(* IEC 61131-3 sources: POMIRTS_lab3/AS/Library_2/AsNxDnS, 3 files *)

(* ---- AsNxDnS.typ ---- *)
TYPE

END_TYPE

(* ---- AsNxDnS.fun ---- *)
{REDUND_CONTEXT} {REDUND_UNREPLICABLE} FUNCTION_BLOCK nxdnsSubscribe			(*subscribe slave*)
	VAR_INPUT
		enable			: BOOL;			(*enables execution*)
		pDevice			: UDINT;		(*interface name given as a pointer, e.g., "SL<x>.SS<y>.IF<z>"*)
	END_VAR
	VAR
        _state			: UINT;			(*internal variable*)
		_result			: UINT;			(*internal variable*)
        _srcId			: UDINT;		(*internal variable*)
	END_VAR
	VAR_OUTPUT
		status			: UINT;			(*execution status: ERR_OK, ERR_FUB_ENABLE_FALSE, ERR_FUB_BUSY, 0xXXXX = see help*)
		dnStatus		: UDINT;		(*devicenet stack status*)
	END_VAR
END_FUNCTION_BLOCK

{REDUND_CONTEXT} {REDUND_UNREPLICABLE} FUNCTION_BLOCK nxdnsUnsubscribe			(*unsubscribe slave*)
	VAR_INPUT
		enable			: BOOL;			(*enables execution*)
		pDevice			: UDINT;		(*interface name given as a pointer, e.g., "SL<x>.SS<y>.IF<z>"*)
	END_VAR
	VAR
        _state			: UINT;			(*internal variable*)
		_result			: UINT;			(*internal variable*)
        _srcId			: UDINT;		(*internal variable*)
	END_VAR
	VAR_OUTPUT
		status			: UINT;			(*execution status: ERR_OK, ERR_FUB_ENABLE_FALSE, ERR_FUB_BUSY, 0xXXXX = see help*)
		dnStatus		: UDINT;		(*devicenet stack status*)
	END_VAR
END_FUNCTION_BLOCK

{REDUND_CONTEXT} {REDUND_UNREPLICABLE} FUNCTION_BLOCK nxdnsRegisterClass		(*register class ID*)
	VAR_INPUT
		enable			: BOOL;			(*enables execution*)
		pDevice			: UDINT;		(*interface name given as a pointer, e.g., "SL<x>.SS<y>.IF<z>"*)
		classId			: UDINT;		(*class designator*)
		accessType		: UDINT;		(*reserved unused, set to 0*)
	END_VAR
	VAR
        _state			: UINT;			(*internal variable*)
		_result			: UINT;			(*internal variable*)
        _srcId			: UDINT;		(*internal variable*)
	END_VAR
	VAR_OUTPUT
		status			: UINT;			(*execution status: ERR_OK, ERR_FUB_ENABLE_FALSE, ERR_FUB_BUSY, 0xXXXX = see help*)
		dnStatus		: UDINT;		(*devicenet stack status*)
	END_VAR
END_FUNCTION_BLOCK

{REDUND_CONTEXT} {REDUND_UNREPLICABLE} FUNCTION_BLOCK nxdnsUnregisterClass		(*unregister class ID*)
	VAR_INPUT
		enable			: BOOL;			(*enables execution*)
		pDevice			: UDINT;		(*interface name given as a pointer, e.g., "SL<x>.SS<y>.IF<z>"*)
		classId			: UDINT;		(*class designator*)
		accessType		: UDINT;		(*reserved unused, set to 0*)
	END_VAR
	VAR
        _state			: UINT;			(*internal variable*)
		_result			: UINT;			(*internal variable*)
        _srcId			: UDINT;		(*internal variable*)
	END_VAR
	VAR_OUTPUT
		status			: UINT;			(*execution status: ERR_OK, ERR_FUB_ENABLE_FALSE, ERR_FUB_BUSY, 0xXXXX = see help*)
		dnStatus		: UDINT;		(*devicenet stack status*)
	END_VAR
END_FUNCTION_BLOCK

{REDUND_CONTEXT} {REDUND_UNREPLICABLE} FUNCTION_BLOCK nxdnsGetAttributeInd		(*get attribute indication*)
	VAR_INPUT
		enable			: BOOL;			(*enables execution*)
		pDevice			: UDINT;		(*interface name given as a pointer, e.g., "SL<x>.SS<y>.IF<z>"*)
	END_VAR
	VAR
        _state			: UINT;			(*internal variable*)
		_result			: UINT;			(*internal variable*)
        _srcId			: UDINT;		(*internal variable*)
	END_VAR
	VAR_OUTPUT
		status			: UINT;			(*execution status: ERR_OK, ERR_FUB_ENABLE_FALSE, ERR_FUB_BUSY, 0xXXXX = see help*)
		dnStatus		: UDINT;		(*devicenet stack status*)
		source			: UDINT;		(*source*)
		sourceId		: UDINT;		(*source ID*)
		classId			: UINT;			(*class ID of user application object requested by master*)
		instanceId		: UINT;			(*instance ID of user application object requested by master*)
		attributeId		: UINT;			(*attribute ID of user application object requested by master*)
	END_VAR
END_FUNCTION_BLOCK

{REDUND_CONTEXT} {REDUND_UNREPLICABLE} FUNCTION_BLOCK nxdnsSetAttributeInd		(*set attribute indication*)
	VAR_INPUT
		enable			: BOOL;			(*enables execution*)
		pDevice			: UDINT;		(*interface name given as a pointer, e.g., "SL<x>.SS<y>.IF<z>"*)
		maxDataCount	: UDINT;		(*maximum data count*)
		pData			: UDINT;		(*information data buffer given as pointer*)
	END_VAR
	VAR
        _state			: UINT;			(*internal variable*)
		_result			: UINT;			(*internal variable*)
        _srcId			: UDINT;		(*internal variable*)
	END_VAR
	VAR_OUTPUT
		status			: UINT;			(*execution status: ERR_OK, ERR_FUB_ENABLE_FALSE, ERR_FUB_BUSY, 0xXXXX = see help*)
		dnStatus		: UDINT;		(*devicenet stack status*)
		source			: UDINT;		(*source*)
		sourceId		: UDINT;		(*source ID*)
		classId			: UINT;			(*class ID of user application object requested by master*)
		instanceId		: UINT;			(*instance ID of user application object requested by master*)
		attributeId		: UINT;			(*attribute ID of user application object requested by master*)
		dataCount		: UINT;			(*data count of bytes to be written by the user application*)
	END_VAR
END_FUNCTION_BLOCK

{REDUND_CONTEXT} {REDUND_UNREPLICABLE} FUNCTION_BLOCK nxdnsGetAttributeRes		(*get attribute response*)
	VAR_INPUT
		enable			: BOOL;			(*enables execution*)
		pDevice			: UDINT;		(*interface name given as a pointer, e.g., "SL<x>.SS<y>.IF<z>"*)
		source			: UDINT;		(*source*)
		sourceId		: UDINT;		(*source ID*)
		classId			: UINT;			(*class ID of user application object requested by master*)
		instanceId		: UINT;			(*instance ID of user application object requested by master*)
		attributeId		: UINT;			(*attribute ID of user application object requested by master*)
		dataCount		: UINT;			(*data count of bytes to be read by the user application*)
		generalError	: USINT;		(*general error code returned by the user, see help*)
		additionalError	: USINT;		(*additional error code, user specific*)
		pData			: UDINT;		(*information data buffer given as pointer*)
	END_VAR
	VAR
        _state			: UINT;			(*internal variable*)
		_result			: UINT;			(*internal variable*)
        _srcId			: UDINT;		(*internal variable*)
	END_VAR
	VAR_OUTPUT
		status			: UINT;			(*execution status: ERR_OK, ERR_FUB_ENABLE_FALSE, ERR_FUB_BUSY, 0xXXXX = see help*)
		dnStatus		: UDINT;		(*devicenet stack status*)
	END_VAR
END_FUNCTION_BLOCK

{REDUND_CONTEXT} {REDUND_UNREPLICABLE} FUNCTION_BLOCK nxdnsSetAttributeRes		(*set attribute response*)
	VAR_INPUT
		enable			: BOOL;			(*enables execution*)
		pDevice			: UDINT;		(*interface name given as a pointer, e.g., "SL<x>.SS<y>.IF<z>"*)
		source			: UDINT;		(*message source*)
		sourceId		: UDINT;		(*message source ID*)
		classId			: UINT;			(*class ID of user application object requested by master*)
		instanceId		: UINT;			(*instance ID of user application object requested by master*)
		attributeId		: UINT;			(*attribute ID of user application object requested by master*)
		dataCount		: UINT;			(*data count of bytes written by the user application*)
		generalError	: USINT;		(*general error code returned by the user, see help*)
		additionalError	: USINT;		(*additional error code, user specific*)
	END_VAR
	VAR
        _state			: UINT;			(*internal variable*)
		_result			: UINT;			(*internal variable*)
        _srcId			: UDINT;		(*internal variable*)
	END_VAR
	VAR_OUTPUT
		status			: UINT;			(*execution status: ERR_OK, ERR_FUB_ENABLE_FALSE, ERR_FUB_BUSY, 0xXXXX = see help*)
		dnStatus		: UDINT;		(*devicenet stack status*)
	END_VAR
END_FUNCTION_BLOCK

{REDUND_CONTEXT} {REDUND_UNREPLICABLE} FUNCTION_BLOCK nxdnsSetAdr				(*set address*)
	VAR_INPUT
		enable			: BOOL;			(*enables execution*)
		pDevice			: UDINT;		(*interface name given as a pointer, e.g., "SL<x>.SS<y>.IF<z>"*)
		address			: UDINT;		(*new slave address*)
	END_VAR
	VAR
        _state			: UINT;			(*internal variable*)
		_result			: UINT;			(*internal variable*)
        _srcId			: UDINT;		(*internal variable*)
	END_VAR
	VAR_OUTPUT
		status			: UINT;			(*execution status: ERR_OK, ERR_FUB_ENABLE_FALSE, ERR_FUB_BUSY, 0xXXXX = see help*)
		dnStatus		: UDINT;		(*devicenet stack status*)
	END_VAR
END_FUNCTION_BLOCK

{REDUND_CONTEXT} {REDUND_UNREPLICABLE} FUNCTION_BLOCK nxdnsStartBusComm		(*start bus communication*)
	VAR_INPUT
		enable			: BOOL;			(*enables execution*)
		pDevice			: UDINT;		(*interface name given as a pointer, e.g., "SL<x>.SS<y>.IF<z>"*)
	END_VAR
	VAR
        _state			: UINT;			(*internal variable*)
		_result			: UINT;			(*internal variable*)
        _srcId			: UDINT;		(*internal variable*)
	END_VAR
	VAR_OUTPUT
		status			: UINT;			(*execution status: ERR_OK, ERR_FUB_ENABLE_FALSE, ERR_FUB_BUSY, 0xXXXX = see help*)
		dnStatus		: UDINT;		(*devicenet stack status*)
	END_VAR
END_FUNCTION_BLOCK

(* ---- AsNxDnS.var ---- *)
VAR CONSTANT
	nxdnsERR_INVALID_DEVICE					: UINT	:= 35360;		(*error invalid device*)
	nxdnsERR_SEND_MESSAGE					: UINT	:= 35361;		(*error send message*)
	nxdnsERR_TIMEOUT						: UINT	:= 35362;		(*error timeout*)
	nxdnsERR_DEVICENET_STACK				: UINT	:= 35363;		(*error receive message*)
	nxdnsERR_PARAMETER						: UINT	:= 35364;		(*error invalid parameter*)
	nxdnsERR_MEMORY							: UINT	:= 35365;		(*error less memory*)
	nxdnsERR_SUBSCRIBE_LISTENER				: UINT	:= 35366;		(*error subscribe listener*)
	nxdnsERR_NO_MORE_ENTRIES				: UINT	:= 35367;		(*error no more entries available*)

	nxdnsGENERR_NO_ERROR					: USINT	:= 16#00;		(*no error*)
	nxdnsGENERR_RES_NOT_AVAIL				: USINT	:= 16#02;		(*resources unavailable, class id invalid*)
	nxdnsGENERR_SERV_NOT_AVAIL				: USINT	:= 16#08;		(*service not available, read or write not supported to class*)
	nxdnsGENERR_ATTRIB_BAD_VALUE			: USINT	:= 16#09;		(*invalid attribute value, attribute not supported*)
	nxdnsGENERR_ATTRIB_NOT_SET				: USINT	:= 16#0E;		(*attribute not settable, attribute has no write permission*)
	nxdnsGENERR_ACCESS_DENIED				: USINT	:= 16#0F;		(*access denied, general error to deny access*)
	nxdnsGENERR_STATE_CONFLICT				: USINT	:= 16#10;		(*state conflict, host state prohibits the command execution*)
	nxdnsGENERR_NOT_ENOUGH_DATA				: USINT	:= 16#13;		(*not enough data received, master has send to less data*)
	nxdnsGENERR_ATTRIB_NOT_SUP				: USINT	:= 16#14;		(*attribute not supported*)
	nxdnsGENERR_TOO_MUCH_DATA				: USINT	:= 16#15;		(*too much data received, master has send to much data*)
	nxdnsGENERR_VENDOR_SPEC_CODE			: USINT	:= 16#1F;		(*vendor specific error code, an addition error code can be placed in additionalError*)
END_VAR
